{attribute 'qualified_only'}
{attribute 'strict'}
TYPE EstadosPrensa :
(
	Parada:=0,
	Entrando,
	Pechando,
	Prensando,
	Aguantando,
	Liberando,
	Abrindo,
	Sacando
);
END_TYPE

(* stored: Version 1.1.0.1, ProductVersion 3.1.4024.11
   DUT EstadosPrensa: Id {dfd9ffef-33db-4a41-936c-6d505dfcba81} *)
